{attribute 'qualified_only'}
VAR_GLOBAL CONSTANT
	MAX_TRAFFIC_LIGHTS: SINT := 4;
END_VAR

(* stored: Version 1.1.0.1, ProductVersion 3.1.4024.12
   GVL GVL: Id {b233d97c-4e18-400a-bd88-a4fa954fb37b} *)
